// TIA Portal project "HMI 2 (butonlar ile sinyal isleme 1)" (V18)

(* hardware
DEVICE "HMI_1"  KTP700 Basic PN
   slot 0: "HMI_1"  KTP700 Basic PN  6AV2 123-2GB03-0AX0  17.0.0.0
   slot 1: "HMI_RT_1"  KTP700 Basic PN  6AV2 123-2GB03-0AX0  17.0.0.0
   slot 5: "HMI_1.IE_CP_1"  PROFINET Interface  17.0.0.0
      slot 1: "PROFINET Interface_1"  PROFINET Interface
         slot 1: "Port_1"  Port
DEVICE "S7-1200 station_1"  S7-1200 Station
   slot 0: "Rack_0"  S7-1200 Rack  Rack  V1.0
   slot 1: "PLC_1"  CPU 1214C AC/DC/Rly  6ES7 214-1BG40-0XB0  V4.6
*)

// ===== PLC "PLC_1"  CPU 1214C AC/DC/Rly =====

VAR_GLOBAL   // PLC tag table "Default tag table"
   "JOG BUTTON" AT %M10.0 : Bool;
   "CIKIS 1" AT %Q0.0 : Bool;
   "START BUT" AT %M10.1 : Bool;
   "STOP BUT" AT %M10.2 : Bool;
   "CIKIS 2" AT %Q0.1 : Bool;
   "TOGGLE BUTTON" AT %M10.3 : Bool;
   "CIKIS 3" AT %Q0.3 : Bool;
END_VAR

ORGANIZATION_BLOCK "Main"   // OB1, LAD, ProgramCycle
TITLE = "Main Program Sweep (Cycle)"
{ S7_Optimized_Access := 'TRUE' }
VERSION : 0.1
   VAR_INPUT
      Initial_Call : Bool;   // Initial call of this OB
      Remanence : Bool;   // =True, if remanent data are available
   END_VAR
BEGIN

REGION Network 1: JOG CALISMA
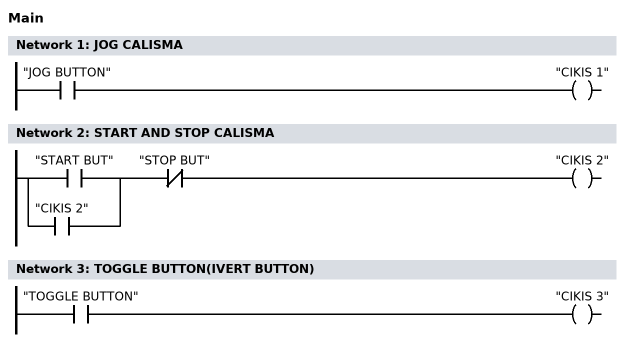
   RUNG wire#powerrail
      Contact( "JOG BUTTON" )
      Coil( "CIKIS 1" )
   END_RUNG
   // the same network as SCL:
   "CIKIS 1" := "JOG BUTTON";
END_REGION

REGION Network 2: START AND STOP CALISMA
   RUNG wire#powerrail
      Contact( "START BUT" )
      wire#w1
      I_Contact( "STOP BUT" )
      Coil( "CIKIS 2" )
   END_RUNG
   RUNG wire#powerrail
      Contact( "CIKIS 2" )
   END_RUNG wire#w1
   // the same network as SCL:
   "CIKIS 2" := ("START BUT" OR "CIKIS 2") AND NOT "STOP BUT";
END_REGION

REGION Network 3: TOGGLE BUTTON(IVERT BUTTON)
   RUNG wire#powerrail
      Contact( "TOGGLE BUTTON" )
      Coil( "CIKIS 3" )
   END_RUNG
   // the same network as SCL:
   "CIKIS 3" := "TOGGLE BUTTON";
END_REGION
END_ORGANIZATION_BLOCK

(* ===== HMI "HMI_RT_1" =====
system functions are stored by id; their names below are inferred from use
connection "HMI_Connection_1": ETHERNET, SMART_S7_1200_OMS

HMI tags "Default tag table"
   "Tag_ScreenNumber" : UInt, internal
   "JOG BUTTON" : Bool = PLC "JOG BUTTON" AT %M10.0, 1 s
   "START BUT" : Bool = PLC "START BUT" AT %M10.1, 1 s
   "STOP BUT" : Bool = PLC "STOP BUT" AT %M10.2, 1 s
   "TOGGLE BUTTON" : Bool = PLC "TOGGLE BUTTON" AT %M10.3, 1 s

screen "Root screen" 800x480
   on GenerateScreen: SetTag("Tag_ScreenNumber", 1)
   TextField "Text field_1" at 308,36 size 202x34; Text 'BUTON TIPLERI'
   Button "Button_1" at 58,122 size 131x51; TextOff 'JOG BUTTON'; TextOn 'JOGGING'
      on Press: SetBit("JOG BUTTON")
      on Release: ResetBit("JOG BUTTON")
   Button "Button_2" at 590,121 size 131x51; TextOff 'STOP BUT'; TextOn 'STOPPED'
      on Press: SetBit("STOP BUT")
      on Release: ResetBit("STOP BUT")
   Button "Button_3" at 430,121 size 131x51; TextOn 'STARTED'; TextOff 'START BUT'
      on Press: SetBit("START BUT")
      on Release: ResetBit("START BUT")
   Button "Button_4" at 56,224 size 131x85; TextOn 'JOGGING'; TextOff 'TOGGLE BUT'
      on Press: InvertBit("TOGGLE BUTTON")
*)